FUNCTION_BLOCK SHAFT_VIEW (* End View of a Rotating Shaft *)
  (* Standard: 61499-1 *)
  (* Version 0.3, 2004-09-01, JHC, Rockwell Automation, Deleted QI,QO; set DIA initial value = 0. *)
  (* Version 0.2, 2001-04-24, JHC, Rockwell Automation, Moved to fb.rt.process. *)
  (* Version 0.1, 2000-06-21, JHC, Rockwell Automation, Uses LibraryElement.dtd *)
  (* Version 0.0, 2000-05-01, JHC, Rockwell Automation *)
  (* Compiler header: package fb.rt.process; *)
  (* Compiler Java IBM VisualAge 3.0 *)
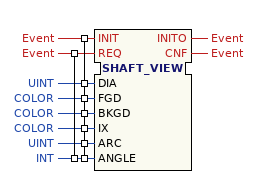
  EVENT_INPUT
    INIT WITH DIA, FGD, BKGD, IX, ARC, ANGLE; (* Initialization *)
    REQ WITH ANGLE; (* Request *)
  END_EVENT
  EVENT_OUTPUT
    INITO; (* Initialization Confirm *)
    CNF; (* Service Confirmation *)
  END_EVENT
  VAR_INPUT
    DIA : UINT; (* Shaft diameter in pixels *)
    FGD : COLOR := COLOR#blue; (* Shaft body color *)
    BKGD : COLOR := COLOR#white; (* Background color *)
    IX : COLOR := COLOR#red; (* Shaft index color *)
    ARC : UINT := 15; (* Shaft mark width *)
    ANGLE : INT; (* Current shaft angle *)
  END_VAR
END_FUNCTION_BLOCK
